(* PLC project BlogProject.project, CODESYS CODESYS V3.5 SP14 Patch 3 *)
(* stored: creationDateTime 2021-10-07T21:06:02.4131783, modificationDateTime 2021-10-07T20:40:20.1109198 *)

FUNCTION_BLOCK mcIsSystemStarted IMPLEMENTS itfEvent
  VAR
    bSystemStarted : BOOL;
  END_VAR

            
          

METHOD getEvent : BOOL
                  getEvent:=bSystemStarted;
                
END_METHOD
END_FUNCTION_BLOCK
